// TIA Portal project "almacen_V16" (V16)

(* hardware
DEVICE "S71500/ET200MP station_1"  S7-1500 station
   slot 0: "Perfil soporte_0"  Rack  6ES7 590-1***0-0AA0
   slot 1: "PLC_1"  CPU 1516-3 PN/DP  6ES7 516-3AN01-0AB0  V2.8
      slot 3: "Display de la CPU_1"  6ES7591-1BA00-0AA0
      slot 32768: "Interfaz PROFINET_1"  X1
      slot 33024: "PROFINET interface_1"  X2
      slot 33280: "DP interface_1"  X3
      slot 34817: "Virtual CP interface port_1"  Virtual CP interface port  Virtual CP interface port
   slot 2: "DI 32x24VDC HF_1"  DI 32x24VDC HF  6ES7 521-1BL00-0AB0  V2.2
   slot 3: "DQ 32x24VDC/0.5A HF_1"  DQ 32x24VDC/0.5A HF  6ES7 522-1BL01-0AB0  V1.1
   slot 4: "AI 8xU/I/RTD/TC ST_1"  AI 8xU/I/RTD/TC ST  6ES7 531-7KF00-0AB0  V2.2
   slot 5: "AQ 4xU/I ST_1"  AQ 4xU/I ST  6ES7 532-5HD00-0AB0  V2.2
DEVICE "Estación PC"  SIMATIC PC station
   slot 0: "Estación PC"  Rail  SIMATIC PC-Station  V1.0
      slot 125: "Stationmanager"  Station_Manager  V6.0.4
   slot 2: "HMI_RT_1"  WinCC RT Advanced  6AV2 104-0xxxx-xxxx  15.1.0.0
      slot 33792: "Interfaz host"  Host interface
   slot 3: "IE general_1"  IE General  IE_CP  V8.2.0
DEVICE "HMI_1"  KTP700 Basic PN
   slot 0: "HMI_1"  KTP700 Basic PN  6AV2 123-2GB03-0AX0  16.0.0.0
   slot 1: "HMI_RT_2"  KTP700 Basic PN  6AV2 123-2GB03-0AX0  16.0.0.0
   slot 5: "HMI_1.IE_CP_1"  PROFINET Interface  16.0.0.0
      slot 1: "PROFINET Interface_1"  PROFINET Interface
         slot 1: "Port_1"  Port
*)

// ===== PLC "PLC_1"  CPU 1516-3 PN/DP =====

VAR_GLOBAL   // PLC tag table "Tabla de variables estándar"
   "STOP" AT %I0.0 : Bool;
   "MARCHA" AT %I0.1 : Bool;
   "LT-01" AT %I0.2 : Bool;
   "EV" AT %Q0.0 : Bool;
   "B-01" AT %Q0.1 : Bool;
   "Limite_superior" AT %Q0.2 : Bool;
   "Nivel_HMI" AT %MD100 : DWord;
   "LSH" AT %IW4 : Int;
   "Frec_HMI" AT %MD104 : DWord;
   "Nivel_cm" AT %MD108 : DWord;
   "Voltios_motor" AT %QW4 : Int;
END_VAR

DATA_BLOCK "Conv_Nivel_DB"   // DB1
{ S7_Optimized_Access := 'TRUE' }
VERSION : 0.1
// stored: InstanceOfName Conv_Nivel
"Conv_Nivel"
BEGIN
END_DATA_BLOCK

DATA_BLOCK "Programa_DB"   // DB2
{ S7_Optimized_Access := 'TRUE' }
VERSION : 0.1
// stored: InstanceOfName Programa
"Programa"
BEGIN
END_DATA_BLOCK

FUNCTION_BLOCK "Conv_Nivel"   // FB1, LAD
{ S7_Optimized_Access := 'TRUE' }
VERSION : 0.1
   VAR_INPUT
      LSH : Int;
      FREC : Int;
   END_VAR
   VAR_OUTPUT
      Nivel_cm : Int;
      Volts : Int;
   END_VAR
   VAR
      LSH_Norm : Real;
      FREC_Norm : Real;
   END_VAR
BEGIN

REGION Network 1
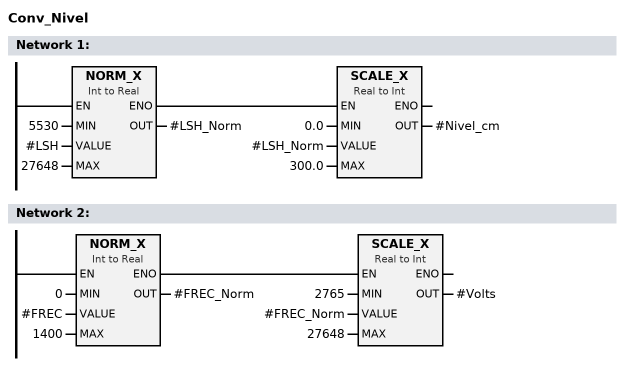
   RUNG wire#powerrail
      { S7_Templates := "[SrcType := Int, DestType := Real]" } Normalize(min := 5530, value := #LSH, max := 27648, out => #LSH_Norm)
      { S7_Templates := "[SrcType := Real, DestType := Int]" } Scale(min := 0.0, value := #LSH_Norm, max := 300.0, out => #Nivel_cm)
   END_RUNG
   // the same network as SCL:
   #LSH_Norm := NORM_X(MIN := 5530, VALUE := #LSH, MAX := 27648);
   #Nivel_cm := SCALE_X(MIN := 0.0, VALUE := #LSH_Norm, MAX := 300.0);
END_REGION

REGION Network 2
   RUNG wire#powerrail
      { S7_Templates := "[SrcType := Int, DestType := Real]" } Normalize(min := 0, value := #FREC, max := 1400, out => #FREC_Norm)
      { S7_Templates := "[SrcType := Real, DestType := Int]" } Scale(min := 2765, value := #FREC_Norm, max := 27648, out => #Volts)
   END_RUNG
   // the same network as SCL:
   #FREC_Norm := NORM_X(MIN := 0, VALUE := #FREC, MAX := 1400);
   #Volts := SCALE_X(MIN := 2765, VALUE := #FREC_Norm, MAX := 27648);
END_REGION
END_FUNCTION_BLOCK

FUNCTION_BLOCK "Programa"   // FB2, LAD
{ S7_Optimized_Access := 'TRUE' }
VERSION : 0.1
   VAR_INPUT
      STOP : Bool;
      MARCHA : Bool;
      "LT-01" : Bool;
      Nivel_sensado : Int;
      Nivel_operador : Int;
   END_VAR
   VAR_OUTPUT
      EV : Bool;
      "B-01" : Bool;
      Limit_Sup : Bool;
   END_VAR
   VAR
      M1 : Bool;
      M2 : Bool;
      M3 : Bool;
      M4 : Bool;
   END_VAR
BEGIN

REGION Network 1
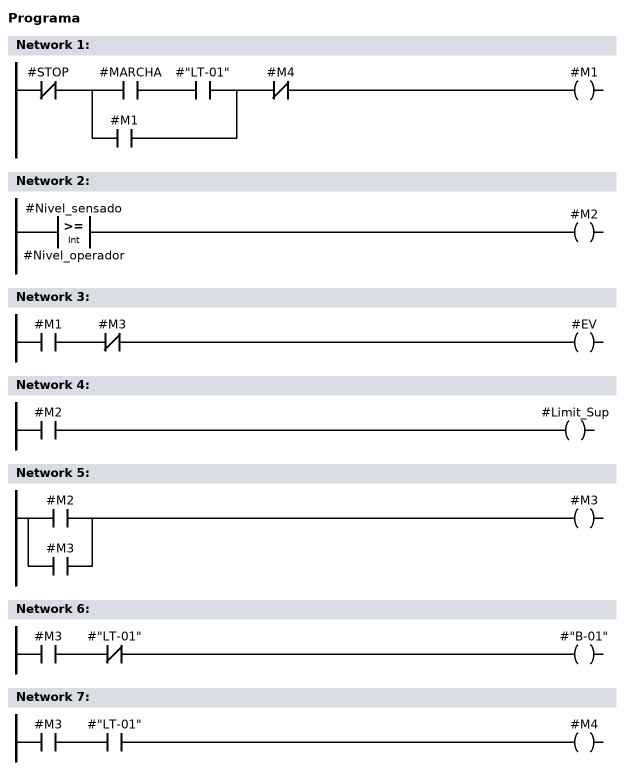
   RUNG wire#powerrail
      I_Contact( #STOP )
      wire#w1
      Contact( #MARCHA )
      Contact( #"LT-01" )
      wire#w2
      I_Contact( #M4 )
      Coil( #M1 )
   END_RUNG
   RUNG wire#w1
      Contact( #M1 )
   END_RUNG wire#w2
   // the same network as SCL:
   #M1 := NOT #STOP AND ((#MARCHA AND #"LT-01") OR #M1) AND NOT #M4;
END_REGION

REGION Network 2
   RUNG wire#powerrail
      { S7_Templates := "SrcType := Int" } GE_Contact(in1 := #Nivel_sensado, in2 := #Nivel_operador)
      Coil( #M2 )
   END_RUNG
   // the same network as SCL:
   #M2 := #Nivel_sensado >= #Nivel_operador;
END_REGION

REGION Network 3
   RUNG wire#powerrail
      Contact( #M1 )
      I_Contact( #M3 )
      Coil( #EV )
   END_RUNG
   // the same network as SCL:
   #EV := #M1 AND NOT #M3;
END_REGION

REGION Network 4
   RUNG wire#powerrail
      Contact( #M2 )
      Coil( #Limit_Sup )
   END_RUNG
   // the same network as SCL:
   #Limit_Sup := #M2;
END_REGION

REGION Network 5
   RUNG wire#powerrail
      Contact( #M2 )
      wire#w1
      Coil( #M3 )
   END_RUNG
   RUNG wire#powerrail
      Contact( #M3 )
   END_RUNG wire#w1
   // the same network as SCL:
   #M3 := #M2 OR #M3;
END_REGION

REGION Network 6
   RUNG wire#powerrail
      Contact( #M3 )
      I_Contact( #"LT-01" )
      Coil( #"B-01" )
   END_RUNG
   // the same network as SCL:
   #"B-01" := #M3 AND NOT #"LT-01";
END_REGION

REGION Network 7
   RUNG wire#powerrail
      Contact( #M3 )
      Contact( #"LT-01" )
      Coil( #M4 )
   END_RUNG
   // the same network as SCL:
   #M4 := #M3 AND #"LT-01";
END_REGION
END_FUNCTION_BLOCK

ORGANIZATION_BLOCK "Main"   // OB1, LAD, ProgramCycle
TITLE = "Main Program Sweep (Cycle)"
{ S7_Optimized_Access := 'TRUE' }
VERSION : 0.1
   VAR_INPUT
      Initial_Call : Bool;   // Initial call of this OB
      Remanence : Bool;   // =True, if remanent data are available
   END_VAR
BEGIN

REGION Network 1
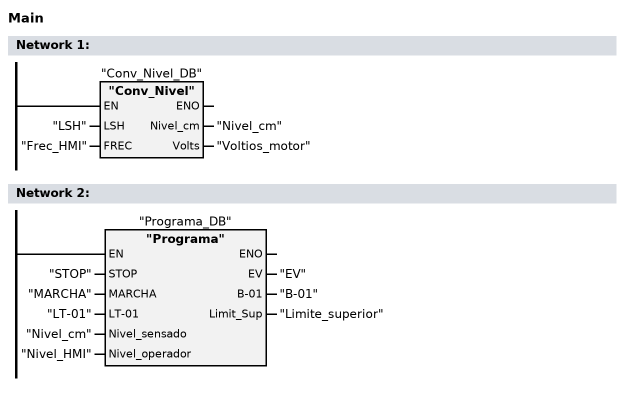
   RUNG wire#powerrail
      "Conv_Nivel_DB"(LSH := "LSH", FREC := "Frec_HMI", Nivel_cm => "Nivel_cm", Volts => "Voltios_motor")
   END_RUNG
   // the same network as SCL:
   "Conv_Nivel_DB"(LSH := "LSH", FREC := "Frec_HMI", Nivel_cm => "Nivel_cm", Volts => "Voltios_motor");   // "Conv_Nivel"
END_REGION

REGION Network 2
   RUNG wire#powerrail
      "Programa_DB"(STOP := "STOP", MARCHA := "MARCHA", "LT-01" := "LT-01", Nivel_sensado := "Nivel_cm", Nivel_operador := "Nivel_HMI", EV => "EV", "B-01" => "B-01", Limit_Sup => "Limite_superior")
   END_RUNG
   // the same network as SCL:
   "Programa_DB"(STOP := "STOP",   // "Programa"
                 MARCHA := "MARCHA",
                 "LT-01" := "LT-01",
                 Nivel_sensado := "Nivel_cm",
                 Nivel_operador := "Nivel_HMI",
                 EV => "EV",
                 "B-01" => "B-01",
                 Limit_Sup => "Limite_superior");
END_REGION
END_ORGANIZATION_BLOCK

(* ===== HMI "HMI_RT_1" =====
system functions are stored by id; their names below are inferred from use
connection "HMI_Connection_2": ETHERNET, S7_1500_OMS

HMI tags "Tabla de variables estándar"
   "Variable_HMI_1" : Int, internal
   "szDataBase" : WString[10], internal
   "szTableName" : WString[10], internal
   "szName_1" : WString[10], internal
   "szName_2" : WString[10], internal
   "sz_Name3" : WString[10], internal
   "nDat_No" : Int, internal
   "nValue_1" : WString[10], internal
   "nValue_2" : Int, internal
   "nValue_3" : Int, internal
   "SearchedName" : WString[10], internal
   "MARCHA" : Bool = PLC MARCHA AT %I0.1, 1 s
   "STOP" : Bool = PLC STOP AT %I0.0, 1 s
   "LT-01" : Bool = PLC "LT-01" AT %I0.2, 1 s
   "EV" : Bool = PLC EV AT %Q0.0, 1 s
   "B-01" : Bool = PLC "B-01" AT %Q0.1, 1 s
   "Nivel_cm" : DWord = PLC Nivel_cm AT %MD108, 1 s
   "Limite_superior" : Bool = PLC Limite_superior AT %Q0.2, 1 s
   "Nivel_HMI" : DWord = PLC Nivel_HMI AT %MD100, 1 s
   "Frec_HMI" : DWord = PLC Frec_HMI AT %MD104, 1 s

screen "crear_borrarDB" 480x640
   TextField "Campo de texto_1" at 36,140 size 107x22; Text 'base de datos'
   IOField "Campo ES_1" at 143,136 size 217x32; FormatPattern ????????????????????
      ProcessValue <- "szDataBase"
   Button "Botón_1" at 167,180 size 165x32; TextOff 'agregar DB'
      on Press: "crear_DB"()
   Button "Botón_2" at 167,221 size 165x32; TextOff 'borrar DB'
      on Press: "borrar_DB"()
   Button "Botón_3" at 352,180 size 96x32; TextOff 'AVISOS'
      on Press: function_ef3f5d25("Ventana de avisos_1", -1)
   Button "Botón_4" at 286,593 size 183x32; TextOff 'control_almacen'
      on Press: ActivateScreen("control_almacen", 0)
   TextField "Campo de texto_2" at 105,16 size 15x22; Text 'Text'
   TextField "Campo de texto_3" at 167,16 size 184x22; Text 'EDICION DE DATA BASE'

screen "control_almacen" 480x640
   Button "Botón_1" at 120,129 size 220x32; TextOff 'crear_borrarDB'
      on Press: ActivateScreen("crear_borrarDB", 0)
   Button "Botón_3" at 120,177 size 220x32; TextOff 'crear|borrar_tablaDB'
      on Press: ActivateScreen("crear_borrartabla", 0)
   TextField "Campo de texto_1" at 154,19 size 157x22; Text 'CONTROL ALMACEN'
   Button "Botón_2" at 120,227 size 220x32; TextOff 'edicion_tablaDB'
      on Press: ActivateScreen("editar_tablaDB", 0)
   Button "Botón_4" at 120,277 size 220x32; TextOff 'edit_data_tablaDB'
      on Press: ActivateScreen("edit_datos_tabla", 0)
   Button "Botón_5" at 120,328 size 220x32; TextOff 'DEL_data_tablaDB'
      on Press: ActivateScreen("eliminar_dato_tabla", 0)
   Button "Botón_6" at 120,377 size 220x32; TextOff 'buscar_data_tablaDB'
      on Press: ActivateScreen("buscar_data_tabla", 0)

screen "crear_borrartabla" 480x640
   TextField "Campo de texto_1" at 10,55 size 192x22; Text 'Nombre de base de datos'
   TextField "Campo de texto_2" at 10,109 size 149x22; Text 'Nombre de la Tabla'
   IOField "Campo ES_1" at 12,77 size 232x32; FormatPattern ????????????????????
      ProcessValue <- "szDataBase"
   Button "Botón_1" at 287,584 size 179x32; TextOff 'Control_almacen'
      on Press: ActivateScreen("control_almacen", 0)
   TextField "Campo de texto_3" at 220,252 size 83x22; Text 'Columna 2'
   TextField "Campo de texto_4" at 220,210 size 83x22; Text 'Columna 1'
   TextField "Campo de texto_5" at 220,296 size 83x22; Text 'Columna 3'
   TextField "Campo de texto_6" at 12,175 size 48x22; Text 'Titulo'
   Button "Botón_2" at 313,77 size 153x32; TextOff 'crear_tabla'
      on Press: "crear_tabla"()
   IOField "Campo ES_2" at 12,134 size 232x32; FormatPattern ????????????????????
      ProcessValue <- "szTableName"
   IOField "Campo ES_3" at 13,200 size 197x32; FormatPattern ??????????
      ProcessValue <- "szName_1"
   IOField "Campo ES_4" at 14,242 size 197x32; FormatPattern ??????????
      ProcessValue <- "szName_2"
   IOField "Campo ES_5" at 13,286 size 198x32; FormatPattern ??????????
      ProcessValue <- "sz_Name3"
   TextField "Campo de texto_7" at 161,14 size 158x22; Text 'DATOS DE TABLA DB'
   Button "Botón_3" at 313,131 size 153x32; TextOff 'borrar_tabla'
      on Press: "borrar_tabla"()

screen "editar_tablaDB" 480x640
   TextField "Campo de texto_1" at 148,15 size 181x22; Text 'EDICION TABLA DATOS'
   Button "Botón_1" at 287,584 size 179x32; TextOff 'Control_almacen'
      on Press: ActivateScreen("control_almacen", 0)
   IOField "Campo ES_1" at 203,67 size 217x32; FormatPattern ????????????????????
      ProcessValue <- "szDataBase"
   TextField "Campo de texto_2" at 1,77 size 192x22; Text 'Nombre de base de datos'
   TextField "Campo de texto_3" at 1,111 size 149x22; Text 'Nombre de la Tabla'
   IOField "Campo ES_2" at 203,101 size 218x32; FormatPattern ????????????????????
      ProcessValue <- "szTableName"
   TextField "Campo de texto_4" at 1,176 size 77x22; Text 'DATO No.'
   IOField "Campo ES_3" at 78,166 size 96x32; FormatPattern s99999
      ProcessValue <- "nDat_No"
   Button "Botón_2" at 191,166 size 131x32; TextOff 'Nuevo Dato'
      on Press: "escribir_dato_tabla"()
   IOField "Campo ES_4" at 78,210 size 246x32; FormatPattern ??????????
      ProcessValue <- "nValue_1"
   TextField "Campo de texto_5" at 1,220 size 58x22; Text 'valor 1'
   TextField "Campo de texto_6" at 1,264 size 59x22; Text 'Valor 2'
   IOField "Campo ES_5" at 78,254 size 96x32; FormatPattern s99999
      ProcessValue <- "nValue_2"
   TextField "Campo de texto_7" at 1,307 size 59x22; Text 'Valor 3'
   IOField "Campo ES_6" at 78,297 size 96x32; FormatPattern s99999
      ProcessValue <- "nValue_3"

screen "edit_datos_tabla" 480x640
   Button "Botón_3" at 372,549 size 99x32; TextOff 'AVISOS'
      on Press: function_ef3f5d25("Ventana de avisos_1", -1)
   Button "Botón_4" at 288,589 size 183x32; TextOff 'control_almacen'
      on Press: ActivateScreen("control_almacen", 0)
   TextField "Campo de texto_3" at 129,16 size 229x22; Text 'EDICION DE DATOS DE TABLA'
   TextField "Campo de texto_1" at 3,83 size 107x22; Text 'base de datos'
   IOField "Campo ES_1" at 159,73 size 217x32; FormatPattern ????????????????????
      ProcessValue <- "szDataBase"
   TextField "Campo de texto_2" at 3,126 size 149x22; Text 'Nombre de la Tabla'
   IOField "Campo ES_2" at 158,116 size 218x32; FormatPattern ????????????????????
      ProcessValue <- "szTableName"
   TextField "Campo de texto_4" at 3,195 size 156x22; Text 'DATO GRABADO No.'
   IOField "Campo ES_3" at 159,185 size 96x32; FormatPattern s99999
      ProcessValue <- "nDat_No"
   Button "Botón_2" at 264,185 size 207x32; TextOff 'reescribir dato'
      on Press: "editar_dato_tabla"()
   TextField "Campo de texto_5" at 20,239 size 31x22; Text 'No.'
   IOField "Campo ES_4" at 65,228 size 199x32; FormatPattern ??????????
      ProcessValue <- "szName_1"
   IOField "Campo ES_5" at 273,228 size 73x32; FormatPattern ??????????
      ProcessValue <- "szName_2"
   IOField "Campo ES_6" at 362,228 size 73x32; FormatPattern ??????????
      ProcessValue <- "sz_Name3"
   IOField "Campo ES_8" at 5,274 size 46x32; FormatPattern s99999
      ProcessValue <- "nDat_No"
   IOField "Campo ES_7" at 65,274 size 199x32; FormatPattern ??????????
      ProcessValue <- "nValue_1"
   IOField "Campo ES_9" at 273,274 size 73x32; FormatPattern s99999
      ProcessValue <- "nValue_2"
   IOField "Campo ES_10" at 362,274 size 73x32; FormatPattern s99999
      ProcessValue <- "nValue_3"

screen "eliminar_dato_tabla" 480x640
   Button "Botón_4" at 288,589 size 183x32; TextOff 'control_almacen'
      on Press: ActivateScreen("control_almacen", 0)
   TextField "Campo de texto_1" at 135,13 size 211x22; Text 'ELIMINACION DATO TABLA'
   TextField "Campo de texto_2" at 3,94 size 107x22; Text 'base de datos'
   IOField "Campo ES_1" at 159,84 size 217x32; FormatPattern ????????????????????
      ProcessValue <- "szDataBase"
   TextField "Campo de texto_3" at 3,137 size 149x22; Text 'Nombre de la Tabla'
   IOField "Campo ES_2" at 158,127 size 218x32; FormatPattern ????????????????????
      ProcessValue <- "szTableName"
   TextField "Campo de texto_4" at 3,206 size 156x22; Text 'DATO GRABADO No.'
   IOField "Campo ES_3" at 159,196 size 96x32; FormatPattern s99999
      ProcessValue <- "nDat_No"
   Button "Botón_2" at 264,196 size 207x32; TextOff 'eliminar dato'
      on Press: "eliminar_dato_tabla"()

screen "buscar_data_tabla" 480x640
   TextField "Campo de texto_3" at 129,16 size 212x22; Text 'BUSCA DE DATOS DE TABLA'
   TextField "Campo de texto_1" at 3,83 size 107x22; Text 'base de datos'
   IOField "Campo ES_1" at 159,73 size 217x32; FormatPattern ????????????????????
      ProcessValue <- "szDataBase"
   TextField "Campo de texto_2" at 3,126 size 149x22; Text 'Nombre de la Tabla'
   IOField "Campo ES_2" at 158,116 size 218x32; FormatPattern ????????????????????
      ProcessValue <- "szTableName"
   TextField "Campo de texto_4" at 3,195 size 156x22; Text 'DATO GRABADO No.'
   IOField "Campo ES_3" at 159,185 size 218x32; FormatPattern ??????????????????????????????
      ProcessValue <- "SearchedName"
   Button "Botón_2" at 158,222 size 220x32; TextOff 'buscar dato'
      on Press: "buscar_dato"()
   TextField "Campo de texto_5" at 24,285 size 31x22; Text 'No.'
   IOField "Campo ES_4" at 69,274 size 199x32; FormatPattern ??????????
      ProcessValue <- "szName_1"
   IOField "Campo ES_5" at 277,274 size 73x32; FormatPattern ??????????
      ProcessValue <- "szName_2"
   IOField "Campo ES_6" at 360,274 size 73x32; FormatPattern ??????????
      ProcessValue <- "sz_Name3"
   IOField "Campo ES_8" at 9,320 size 46x32; FormatPattern s99999
      ProcessValue <- "nDat_No"
   IOField "Campo ES_7" at 69,320 size 199x32; FormatPattern ??????????
      ProcessValue <- "nValue_1"
   IOField "Campo ES_9" at 277,320 size 73x32; FormatPattern s99999
      ProcessValue <- "nValue_2"
   IOField "Campo ES_10" at 360,320 size 73x32; FormatPattern s99999
      ProcessValue <- "nValue_3"
   Button "Botón_4" at 288,589 size 183x32; TextOff 'control_almacen'
      on Press: ActivateScreen("control_almacen", 0)
   AlarmView "Visor de avisos_1" at 0,352 size 480x18

screen "Screen_1" 480x640
   IOField "I/O field_1" at 271,140 size 96x32; FormatPattern s999
      ProcessValue <- "Nivel_HMI"
   TextField "Text field_2" at 140,140 size 111x23; Text 'Setpoint (cm) / Setpoint(cm)'
   Circle "Circle_1" at 152,336 size 48x48
      Appearance <- "EV"
   Circle "Circle_2" at 241,336 size 48x48
      Appearance <- "B-01"
   TextField "Text field_6" at 160,394 size 26x23; Text 'EV'
   TextField "Text field_7" at 246,391 size 43x23; Text 'Bomba / B-01'
   GraphicView "Graphic view_1" at 108,262 size 116x65; Picture "Graphic_2"
   IOField "I/O field_2" at 271,176 size 96x32; FormatPattern s999
      ProcessValue <- "Frec_HMI"
   TextField "Text field_1" at 140,185 size 84x23; Text 'Setpoint (cm) / Velocidad'
   Circle "Circle_4" at 27,336 size 48x48
      Appearance <- "LT-01"
   TextField "Text field_3" at 27,394 size 52x23; Text 'EV / LT-01'
   Button "Button_3" at 25,505 size 96x32; TextOff 'Guardar'
      on Release: "WriteToExcel"()
   Circle "Circle_3" at 246,463 size 48x48
      Appearance <- "Limite_superior"
   TextField "Text field_4" at 201,529 size 128x23; Text 'Limite superior'
   Button "Button_1" at 9,140 size 96x32; TextOff 'MARCHA / Marcha'
      on Release: ResetBit("MARCHA")
      on Press: SetBit("MARCHA")
      Appearance <- "MARCHA"
   Button "Button_2" at 6,184 size 96x32; TextOff 'PARO / Paro'
      on Release: ResetBit("STOP")
      on Press: SetBit("STOP")
      Appearance <- "STOP"
   Bar "Bar_1" at 375,283 size 85x228; MinimumValue 0; MaximumValue 300
      ProcessValue <- "Nivel_cm"
   Button "Button_4" at 27,445 size 96x32; TextOff 'Runtime'
      on Release: StopRuntime(0)

VB script "crear_DB"
   'declaracion de variables locales
   Dim conn, rst, BDatos
   On Error Resume Next
   'el objeto ADODB. Connection permite conectarse a una base de datos
   'el objeto ADODB.Recordset contendra el resultado de la solicitud.
   Set conn = CreateObject ("ADODB.Connection")
   Set rst = CreateObject ("ADODB.Recordset")
   
   'conn.open abre conexion
   'provide especifica el proveedor OLE
   'MSDASQL permite que las aplicaciones del cliente de OLE DB
   'usen controladores ODBC para conectarse a una fuente de datos
   
   'Database_1 es un tipo ODBC
   
   conn.open "Provider=MSDASQL; DSN=Database_1"
   
   'rutina de error
   If Err.Number <>0 Then
   	bfde4b54-0db7-4817-8032-87127bf19bb9 "Error #" & Err.Number & " " & Err.Description
   	Err.Clear
   	Exit Sub
   End If
   
   'definicion de nueva base de datos
   BDatos = "CREATE DATABASE " & SmartTags("szDataBase")
   
   'crea la nueva base de datos
   Set rst = conn.Execute(BDatos)
   
   'rutina de error
   If Err.Number <>0 Then
   	bfde4b54-0db7-4817-8032-87127bf19bb9 "Error #" & Err.Number & " " & Err.Description
   	Err.Clear
   	Exit Sub
   End If
   
   'cierra conexion
   conn.close
   Set conn = Nothing
   Set rst = Nothing
   	

VB script "borrar_DB"
   'declaracion de variables locales
   Dim conn, rst, BDatos
   On Error Resume Next
   'el objeto ADODB. Connection permite conectarse a una base de datos
   'el objeto ADODB.Recordset contendra el resultado de la solicitud.
   Set conn = CreateObject ("ADODB.Connection")
   Set rst = CreateObject ("ADODB.Recordset")
   
   'conn.open abre conexion
   'provide especifica el proveedor OLE
   'MSDASQL permite que las aplicaciones del cliente de OLE DB
   'usen controladores ODBC para conectarse a una fuente de datos
   
   'Database_1 es un tipo ODBC
   
   conn.open "Provider=MSDASQL; DSN=Database_1"
   
   'rutina de error
   If Err.Number <>0 Then
   	bfde4b54-0db7-4817-8032-87127bf19bb9 "Error #" & Err.Number & " " & Err.Description
   	Err.Clear
   	Exit Sub
   End If
   
   'definicion de nueva base de datos
   BDatos = "DROP DATABASE " & SmartTags("szDataBase")
   
   'crea la nueva base de datos
   Set rst = conn.Execute(BDatos)
   
   'rutina de error
   If Err.Number <>0 Then
   	bfde4b54-0db7-4817-8032-87127bf19bb9 "Error #" & Err.Number & " " & Err.Description
   	Err.Clear
   	Exit Sub
   End If
   
   'cierra conexion
   conn.close
   Set conn = Nothing
   Set rst = Nothing

VB script "crear_tabla"
   'declaracion de variables locales
   Dim conn, rst, BDatos
   On Error Resume Next
   'el objeto ADODB. Connection permite conectarse a una base de datos
   'el objeto ADODB.Recordset contendra el resultado de la solicitud.
   Set conn = CreateObject ("ADODB.Connection")
   Set rst = CreateObject ("ADODB.Recordset")
   
   'conn.open abre conexion
   'provide especifica el proveedor OLE
   'MSDASQL permite que las aplicaciones del cliente de OLE DB
   'usen controladores ODBC para conectarse a una fuente de datos
   
   'Database_1 es un tipo ODBC
   'Initial Catalog es el nombre de la base de datos que utilizara la cadena de conexion
   
   conn.Open "Provider=MSDASQL;Initial Catalog=" & SmartTags("szDataBase") & _
   ";DSN=S7PLCDB"
             
   'rutina de error
   If Err.Number <>0 Then
   	bfde4b54-0db7-4817-8032-87127bf19bb9 "Error #" & Err.Number & " " & Err.Description
   	Err.Clear
   	Exit Sub
   End If
   
   'SMALLINT tipo de datos de 16 bits ocupan poco espacio de memoria
   'definicion de SQL tabla
   
   BDatos = "CREATE TABLE "& SmartTags("szTableName") & " (Nr SMALLINT,"  _ 
   			& SmartTags("szName_1") & " CHAR (30), " & SmartTags("szName_2") & " SMALLINT, "_ 
   			& SmartTags("sz_Name3") & " SMALLINT)"
    
    
   'crea la nueva base de datos
   Set rst = conn.Execute(BDatos)
   
   'rutina de error
   If Err.Number <>0 Then
   	bfde4b54-0db7-4817-8032-87127bf19bb9 "Error #" & Err.Number & " " & Err.Description
   	Err.Clear
   	Exit Sub
   End If
   
   'cierra conexion
   conn.close
   Set conn = Nothing
   Set rst = Nothing
   	

VB script "borrar_tabla"
   'declaracion de variables locales
   Dim conn, rst, BDatos
   On Error Resume Next
   'el objeto ADODB. Connection permite conectarse a una base de datos
   'el objeto ADODB.Recordset contendra el resultado de la solicitud.
   Set conn = CreateObject ("ADODB.Connection")
   Set rst = CreateObject ("ADODB.Recordset")
   
   'conn.open abre conexion
   'provide especifica el proveedor OLE
   'MSDASQL permite que las aplicaciones del cliente de OLE DB
   'usen controladores ODBC para conectarse a una fuente de datos
   
   'Database_1 es un tipo ODBC
   'Initial Catalog es el nombre de la base de datos que utilizara la cadena de conexion
   
   conn.Open "Provider=MSDASQL;Initial Catalog=" & SmartTags("szDataBase") & _
   ";DSN=Database_1"
             
   'rutina de error
   If Err.Number <>0 Then
   	bfde4b54-0db7-4817-8032-87127bf19bb9 "Error #" & Err.Number & " " & Err.Description
   	Err.Clear
   	Exit Sub
   End If
   
   'BORRADO DE DATOS DE TABLA
   BDatos = "DROP TABLE "& SmartTags("szTableName") 
    
    
   'crea la nueva base de datos
   Set rst = conn.Execute(BDatos)
   
   'rutina de error
   If Err.Number <>0 Then
   	bfde4b54-0db7-4817-8032-87127bf19bb9 "Error #" & Err.Number & " " & Err.Description
   	Err.Clear
   	Exit Sub
   End If
   
   'cierra conexion
   conn.close
   Set conn = Nothing
   Set rst = Nothing

VB script "escribir_dato_tabla"
   'declaracion de variables locales
   Dim conn, rst, BDatos
   On Error Resume Next
   'el objeto ADODB. Connection permite conectarse a una base de datos
   'el objeto ADODB.Recordset contendra el resultado de la solicitud.
   Set conn = CreateObject ("ADODB.Connection")
   Set rst = CreateObject ("ADODB.Recordset")
   
   'conn.open abre conexion
   'provide especifica el proveedor OLE
   'MSDASQL permite que las aplicaciones del cliente de OLE DB
   'usen controladores ODBC para conectarse a una fuente de datos
   
   'Database_1 es un tipo ODBC
   'Initial Catalog es el nombre de la base de datos que utilizara la cadena de conexion
   
   conn.Open "Provider=MSDASQL;Initial Catalog=" & SmartTags("szDataBase") & _
   ";DSN=Database_1"
             
   'rutina de error
   If Err.Number <>0 Then
   	bfde4b54-0db7-4817-8032-87127bf19bb9 "Error #" & Err.Number & " " & Err.Description
   	Err.Clear
   	Exit Sub
   End If
   
   'seleccionar registro de datos de la tabla (donde Nr = nDat_No)
   '* = Todos los datos
   
   BDatos = "SELECT * FROM " & SmartTags("szTableName") & " WHERE Nr = " & SmartTags("nDat_No")
   
   'crea la nueva base de datos
   Set rst = conn.Execute(BDatos)
   
   'rutina de error
   If Err.Number <>0 Then
   	bfde4b54-0db7-4817-8032-87127bf19bb9 "Error #" & Err.Number & " " & Err.Description
   	Err.Clear
   	Exit Sub
   End If
   
   'comprobar si el registro de datos tiene datos dentro de la tabla
   If Not(rst.EOF And rst.BOF) Then
   	bfde4b54-0db7-4817-8032-87127bf19bb9 "Ya existe dato guardado en tabla"
   	rst.Close
   Else
   	'definicion de registro de datos
   	BDatos = "INSERT INTO " & SmartTags("szTableName") & " VALUES ('" & SmartTags("nDat_No") & _
   	"' , '" & SmartTags("nValue_1") & "' , '" & SmartTags("nValue_2") & _
   	"' , '" & SmartTags("nValue_3") & "')"
   
   'insertar registro de datos de la tabla
   Set rst=conn.Execute(BDatos)
   
   End If
   'cierra conexion
   conn.close
   Set conn = Nothing
   Set rst = Nothing

VB script "editar_dato_tabla"
   'declaracion de variables locales
   Dim conn, rst, BDatos
   On Error Resume Next
   'el objeto ADODB. Connection permite conectarse a una base de datos
   'el objeto ADODB.Recordset contendra el resultado de la solicitud.
   Set conn = CreateObject ("ADODB.Connection")
   Set rst = CreateObject ("ADODB.Recordset")
   
   'conn.open abre conexion
   'provide especifica el proveedor OLE
   'MSDASQL permite que las aplicaciones del cliente de OLE DB
   'usen controladores ODBC para conectarse a una fuente de datos
   
   'Database_1 es un tipo ODBC
   'Initial Catalog es el nombre de la base de datos que utilizara la cadena de conexion
   
   conn.Open "Provider=MSDASQL;Initial Catalog=" & SmartTags("szDataBase") & _
   ";DSN=Database_1"
             
   'rutina de error
   If Err.Number <>0 Then
   	bfde4b54-0db7-4817-8032-87127bf19bb9 "Error #" & Err.Number & " " & Err.Description
   	Err.Clear
   	Exit Sub
   End If
   
   'seleccionar registro de datos de la tabla (donde Nr = nDat_No)
   '* = Todos los datos
   
   BDatos = "SELECT * FROM " & SmartTags("szTableName") & " WHERE Nr = " & SmartTags("nDat_No")
   
   'crea la nueva base de datos
   Set rst = conn.Execute(BDatos)
   
   'rutina de error
   If Err.Number <>0 Then
   	bfde4b54-0db7-4817-8032-87127bf19bb9 "Error #" & Err.Number & " " & Err.Description
   	Err.Clear
   	Exit Sub
   End If
   
   'comprobar si el rst viene vacio. si tiene contenido, se muestra
   If Not (rst.EOF And rst.BOF) Then
   	
   	rst.MoveFirst 'mueve el puntero al primer registro
   	
   	SmartTags("szName_1") = rst.Fields(1).Name
   	SmartTags("szName_2") = rst.Fields(2).Name
   	SmartTags("sz_Name3") = rst.Fields(3).Name
   	
   	rst.close
   Else
   	bfde4b54-0db7-4817-8032-87127bf19bb9 "El dato buscado no esta disponible"
   End If
   
   'definicion de datos grabados
   BDatos = "UPDATE " & SmartTags("szTableName") & " Set " & SmartTags("szName_1") & " = '" & SmartTags("nValue_1") & "' , " & SmartTags("szName_2") & " = " & SmartTags("nValue_2") & " , " & SmartTags("sz_Name3") & " = " & SmartTags("nValue_3") & " WHERE Nr = " & SmartTags("nDat_No")
   
   'actualizar data guardada 
   Set rst = conn.Execute(BDatos)
   
   'Error de rutina
   If Err.Number <> 0 Then
   	bfde4b54-0db7-4817-8032-87127bf19bb9 "Error #" & Err.Number & " " & Err.Description
   	Err.Clear
   	Exit Sub
   End If
   
   'cierra conexion
   conn.close
   Set conn = Nothing
   Set rst = Nothing

VB script "eliminar_dato_tabla"
   'declaracion de variables locales
   Dim conn, rst, BDatos
   On Error Resume Next
   'el objeto ADODB. Connection permite conectarse a una base de datos
   'el objeto ADODB.Recordset contendra el resultado de la solicitud.
   Set conn = CreateObject ("ADODB.Connection")
   Set rst = CreateObject ("ADODB.Recordset")
   
   'conn.open abre conexion
   'provide especifica el proveedor OLE
   'MSDASQL permite que las aplicaciones del cliente de OLE DB
   'usen controladores ODBC para conectarse a una fuente de datos
   
   'Database_1 es un tipo ODBC
   'Initial Catalog es el nombre de la base de datos que utilizara la cadena de conexion
   
   conn.Open "Provider=MSDASQL;Initial Catalog=" & SmartTags("szDataBase") & _
   ";DSN=Database_1"
             
   'rutina de error
   If Err.Number <>0 Then
   	bfde4b54-0db7-4817-8032-87127bf19bb9 "Error #" & Err.Number & " " & Err.Description
   	Err.Clear
   	Exit Sub
   End If
   
   'seleccionar registro de datos de la tabla (donde Nr = nDat_No)
   '* = Todos los datos
   
   BDatos = "DELETE FROM " & SmartTags("szTableName") & " WHERE Nr = " & SmartTags("nDat_No")
   
   'elimina el dato de la tabla
   Set rst = conn.Execute(BDatos)
   
   'rutina de error
   If Err.Number <>0 Then
   	bfde4b54-0db7-4817-8032-87127bf19bb9 "Error #" & Err.Number & " " & Err.Description
   	Err.Clear
   	Exit Sub
   End If
   
   'cierra conexion
   conn.close
   Set conn = Nothing
   Set rst = Nothing

VB script "buscar_dato"
   Dim conn, rst, BDatos, nombre,SearchedName ', val1, val2, val3   'Declaracion de variables locales
   nombre= SmartTags("szName_1") 
   SearchedName= SmartTags("SearchedName")
   'val1= SmartTags("valor1_nombre")
   'val2= SmartTags("valor2_px")
   'val3= SmartTags("valor3_py")
   
   On Error Resume Next   'Activa el tratamiento de errores 
   
   'El objeto ADODB.Connection permite establecer un vínculo con la base de datos
   'El objecto ADODB.Recordset servir par la manipulación de datos.
   Set conn = CreateObject ("ADODB.Connection")
   Set rst = CreateObject ("ADODB.Recordset")
   
   'conn.Open = Abre conexion
   'Provider = especifica el proveedor OLE
   'MSDASQL = Permite que las aplicaciones del cliente de OLE DB
   '          usen controladores ODBC para conectarse a una fuente de datos
   'Initial Catalog = Es el nombre de la base de datos que utilizará la cadena de conexión.
   'Database_1 = Fuente de datos tipo ODBC
   conn.Open "Provider=MSDASQL;Initial Catalog =" & SmartTags("szDataBase") & _
             ";DSN=Database_1"
   
   'rutina de error
   If Err.Number <>0 Then
   	bfde4b54-0db7-4817-8032-87127bf19bb9 "Error #" & Err.Number & " " & Err.Description
   	Err.Clear
   	Exit Sub
   End If
   
   'Seleccionar registro de datos de la tabla (donde Nr = nDat_No) 
   '   * = todos los datos
   'BDatos = "SELECT * FROM " & SmartTags("szTableName") & " WHERE  name = " & SmartTags("nValue_1") 
   'Escribe un registro de datos en una tabla.
   'BDatos = "SELECT  nombre FROM  Datos   WHERE  nombre = "& SmartTags("nValue_1")
    BDatos = "SELECT * FROM " & SmartTags("szTableName") & " WHERE  nombre LIKE " & "'" & SearchedName &  "'"
   
   Set rst = conn.Execute(BDatos)
   
   'Error routine - Fehler Routine
   If Err.Number <> 0 Then
   	bfde4b54-0db7-4817-8032-87127bf19bb9 "Error #" & Err.Number & " " & Err.Description
   	Err.Clear 
   	Exit Sub
   End If
   
   'Se comprueba si rst viene vacio. Si tiene contenido, se muestra
   If Not (rst.EOF And rst.BOF) Then 
   	
   	rst.MoveFirst 'mueve el puntero al primer registro
   	SmartTags("nDat_No") = rst.Fields(0).Value 
   	SmartTags("nValue_1") = rst.Fields(1).Value
   	SmartTags("nValue_2") = rst.Fields(2).Value
   	SmartTags("nValue_3") = rst.Fields(3).Value
   	SmartTags("szName_1") = rst.Fields(1).Name
   	SmartTags("szName_2") = rst.Fields(2).Name
   	SmartTags("sz_Name3") = rst.Fields(3).Name 
   	
   	rst.close 
   Else
   	bfde4b54-0db7-4817-8032-87127bf19bb9 "El dato buscado no esta disponible" 
   End If
   
   'Se cierran los objetos que se abrieron
   conn.close
   
   'se liberan los recursos que el servidor les habia asignado con la instrucción Nothing.
   Set conn= Nothing
   Set rst = Nothing

VB script "WriteToExcel"
   'Tip:
   ' 1. Use the <CTRL+SPACE> or <CTRL+I> shortcut to open a list of all objects and functions
   ' 2. Write the code using the HMI Runtime object.
   '  Example: HmiRuntime.Screens("Screen_1").
   ' 3. Use the <CTRL+J> shortcut to create an object reference.
   'Write the code as of this position:
   Dim FolderWay, ObjectWay, FileName, File, FileExist, Apendix, Row
   
   FolderWay = "C:\Test\Database"
   
   Set ObjectWay = CreateObject("Scripting.FileSystemObject")
   
   If Not ObjectWay.FolderExists(FolderWay) Then
   	ObjectWay.CreateFolder FolderWay
   End If
   
   FileName = "Datos.csv"
   Set File = CreateObject("Scripting.FileSystemObject")
   
   FileExist = File.FileExists(FolderWay & "\" & FileName)
   
   If FileExist=False Then
   	File.CreateTextFile(FolderWay & "\" & FileName)
   	Set Apendix = File.OpenTextFile(FolderWay & "\" & FileName,4)
   	Apendix.WriteLine(" Data 1; Data 2")
   	Apendix.Close
   	
   	Set File = Nothing
   	
   End If
   
   Set File = CreateObject("Scripting.FileSystemObject")
   Set Row = File.OpenTextFile(FolderWay & "\" & FileName,4)
   
   Row.WriteLine("Integer" & ";" & "Integer")
   Row.Close
*)

(* ===== HMI "HMI_RT_2" =====
system functions are stored by id; their names below are inferred from use
connection "HMI_Connection_1": ETHERNET, SMART_S7_1500_OMS

HMI tags "Default tag table"
   "Tag_ScreenNumber" : UInt, internal
   "MARCHA" : Bool = PLC MARCHA AT %I0.1, 1 s
   "STOP" : Bool = PLC STOP AT %I0.0, 1 s
   "EV" : Bool = PLC EV AT %Q0.0, 1 s
   "B-01" : Bool = PLC "B-01" AT %Q0.1, 1 s
   "Limite_superior" : Bool = PLC Limite_superior AT %Q0.2, 1 s
   "Nivel_cm" : DWord = PLC Nivel_cm AT %MD108, 1 s
   "Frec_HMI" : DWord = PLC Frec_HMI AT %MD104, 1 s
   "Nivel_HMI" : DWord = PLC Nivel_HMI AT %MD100, 1 s
   "LT-01" : Bool = PLC "LT-01" AT %I0.2, 1 s

text list "Nombre_imagen_lista_texto": 1 'Root screen'; 2 'Proceso'; 3 'Imágenes de sistema'; 4 'Información del proyecto'; 5 'Administración de usuarios'; 6 'Información de sistema'

Template "Template_1" 800x480
   Button "Salir" at 714,429 size 71x50; TextOff 'Salir'; PictureOff "ExitRuntime_KTP700_Basic_PN_TR"; PictureOn "ExitRuntime_KTP700_Basic_PN_TR"
      on Release: StopRuntime(0)
   Button "Template_Button" at 614,429 size 71x50; TextOff 'Text'
   Button "Template_Button_1" at 514,429 size 71x50; TextOff 'Text'
   Button "Template_Button_2" at 414,429 size 71x50; TextOff 'Text'
   Button "Template_Button_3" at 314,429 size 71x50; TextOff 'Text'
   Button "Template_Button_4" at 214,429 size 71x50; TextOff 'Text'
   Button "Avisos" at 114,429 size 71x50; TextOff 'Avisos'; PictureOff "AlarmDisplay_KTP700_Basic_PN_TR"; PictureOn "AlarmDisplay_KTP700_Basic_PN_TR"
      on Release: function_ef3f5d25("Alarm window_Unacknowledged", -1)
   Button "Imagen inicial" at 14,429 size 71x50; TextOff 'Imagen inicial'; PictureOff "NavigateHome_KTP700_Basic_PN_TR"; PictureOn "NavigateHome_KTP700_Basic_PN_TR"
      on Release: ActivateScreen("Root screen", 0)
   SymbolicIOField "Symbolic_IO_Field_Screen" at 93,9 size 600x33; TextOff '0'; TextOn '1'; TextList "Nombre_imagen_lista_texto"
      ProcessValue <- "Tag_ScreenNumber"
      on Change: ActivateScreenByNumber("Tag_ScreenNumber", 0)
   DateTimeField "HmiScreenItemData" at 695,25 size 105x25
   DateTimeField "HmiScreenItemData_1" at 695,0 size 105x25
   GraphicView "Logotipo" at 0,0 size 91x51; Picture "Logotipo de HMI_1"

screen "Root screen" 800x480, template "Template_1"
   on GenerateScreen: SetTag("Tag_ScreenNumber", 1)
   TextField "HmiScreenItemData_1" at 80,225 size 640x25; Text 'Bienvenido a HMI_1 (KTP700 Basic+ PN)!'
   Button "HmiScreenItemData" at 36,87 size 159x47; TextOff 'Proceso'; PictureOff "Navigates to Proceso for KTP700 Basic+ PN 16.0.0.0"; PictureOn "Navigates to Proceso for KTP700 Basic+ PN 16.0.0.0"
      on Release: ActivateScreen("Proceso", 0)
   Button "HmiScreenItemData_2" at 36,146 size 159x47; TextOff 'Imágenes de sistema'; PictureOff "Navigates to System screens for KTP700 Basic+ PN 16.0.0.0"; PictureOn "Navigates to System screens for KTP700 Basic+ PN 16.0.0.0"
      on Release: ActivateScreen("System screens", 0)

screen "Proceso" 800x480, template "Template_1"
   on GenerateScreen: SetTag("Tag_ScreenNumber", 2)
   TextField "HmiScreenItemData" at 33,83 size 640x25; Text 'Proceso'
   Button "Atrás" at 1,52 size 159x47; TextOff 'Atrás'
      on Release: ActivateScreen("Root screen", 0)
   Button "Button_1" at 66,159 size 96x32; TextOff 'MARCHA / Marcha'
      on Release: ResetBit("MARCHA")
      on Press: SetBit("MARCHA")
      Appearance <- "MARCHA"
   Button "Button_2" at 66,212 size 96x32; TextOff 'PARO / Paro'
      on Release: ResetBit("STOP")
      on Press: SetBit("STOP")
      Appearance <- "STOP"
   IOField "I/O field_1" at 383,138 size 96x32; FormatPattern s999
      ProcessValue <- "Nivel_HMI"
   TextField "Text field_2" at 225,140 size 111x23; Text 'Setpoint (cm) / Setpoint(cm)'
   Circle "Circle_1" at 301,327 size 48x48
      Appearance <- "EV"
   Circle "Circle_2" at 433,327 size 48x48
      Appearance <- "B-01"
   Circle "Circle_3" at 567,327 size 48x48
      Appearance <- "Limite_superior"
   TextField "Text field_4" at 531,389 size 128x23; Text 'Limite superior'
   TextField "Text field_6" at 310,384 size 26x23; Text 'EV'
   TextField "Text field_7" at 433,387 size 43x23; Text 'Bomba / B-01'
   GraphicView "Graphic view_1" at 301,255 size 116x65; Picture "Graphic_2"
   IOField "I/O field_2" at 383,187 size 96x32; FormatPattern s999
      ProcessValue <- "Frec_HMI"
   TextField "Text field_1" at 225,189 size 84x23; Text 'Setpoint (cm) / Velocidad'
   Bar "Bar_1" at 670,163 size 85x228; MinimumValue 0; MaximumValue 300
      ProcessValue <- "Nivel_cm"
   TextField "Text field_5" at 639,138 size 138x23; Text 'Nivel tanque / Nivel del tanque'
   Circle "Circle_4" at 67,320 size 48x48
      Appearance <- "LT-01"
   TextField "Text field_3" at 67,378 size 52x23; Text 'EV / LT-01'

screen "System screens" 800x480, template "Template_1"
   on GenerateScreen: SetTag("Tag_ScreenNumber", 3)
   Button "Atrás" at 1,52 size 159x47; TextOff 'Atrás'
      on Release: ActivateScreen("Root screen", 0)
   Button "HmiScreenItemData" at 36,146 size 159x47; TextOff 'Información del proyecto'; PictureOff "Navigates to Project information for KTP700 Basic+ PN 16.0.0.0"; PictureOn "Navigates to Project information for KTP700 Basic+ PN 16.0.0.0"
      on Release: ActivateScreen("Project information", 0)
   Button "HmiScreenItemData_1" at 36,205 size 159x47; TextOff 'Administración de usuarios'; PictureOff "Navigates to User administration for KTP700 Basic+ PN 16.0.0.0"; PictureOn "Navigates to User administration for KTP700 Basic+ PN 16.0.0.0"
      on Release: ActivateScreen("User administration", 0)
   Button "HmiScreenItemData_2" at 36,264 size 159x47; TextOff 'Información de sistema'; PictureOff "Navigates to System information for KTP700 Basic+ PN 16.0.0.0"; PictureOn "Navigates to System information for KTP700 Basic+ PN 16.0.0.0"
      on Release: ActivateScreen("System information", 0)

screen "Project information" 800x480, template "Template_1"
   on GenerateScreen: SetTag("Tag_ScreenNumber", 4)
   TextField "HmiScreenItemData" at 35,102 size 171x28; Text 'Nombre del proyecto:'
   TextField "HmiScreenItemData_1" at 241,102 size 524x28; Text 'almacen_V16'
   TextField "HmiScreenItemData_2" at 35,132 size 171x28; Text 'Creado:'
   TextField "HmiScreenItemData_3" at 241,132 size 524x28; Text '10/27/2021 3:28:15 PM'
   TextField "HmiScreenItemData_4" at 35,162 size 171x28; Text 'Autor:'
   TextField "HmiScreenItemData_5" at 241,162 size 524x28; Text 'adria'
   TextField "HmiScreenItemData_6" at 35,192 size 171x28; Text 'Descripción:'
   TextField "HmiScreenItemData_7" at 241,192 size 524x28; Text '(no configurado)'
   Button "Atrás" at 1,52 size 159x47; TextOff 'Atrás'
      on Release: ActivateScreen("System screens", 0)

screen "User administration" 800x480, template "Template_1"
   on GenerateScreen: SetTag("Tag_ScreenNumber", 5)
   UserView "HmiScreenItemData" at 1,100 size 796x321
   Button "Atrás" at 1,52 size 159x47; TextOff 'Atrás'
      on Release: ActivateScreen("System screens", 0)

screen "System information" 800x480, template "Template_1"
   on GenerateScreen: SetTag("Tag_ScreenNumber", 6)
   TextField "HmiScreenItemData" at 35,102 size 171x28; Text 'Tipo de panel:'
   TextField "HmiScreenItemData_1" at 241,102 size 524x28; Text 'KTP700 Basic+ PN 16.0.0.0'
   TextField "HmiScreenItemData_2" at 35,132 size 171x28; Text 'Conexión:'
   TextField "HmiScreenItemData_3" at 241,132 size 524x28; Text 'PROFINET (X1)'
   TextField "HmiScreenItemData_4" at 35,162 size 171x28; Text 'Controlador:'
   TextField "HmiScreenItemData_5" at 241,162 size 524x28; Text 'SIMATIC S7 1500'
   Button "Atrás" at 1,52 size 159x47; TextOff 'Atrás'
      on Release: ActivateScreen("System screens", 0)
*)